Fanuc KAREL source: kb00151.KL

-- PROVISIONAL review KL for V940-1; original PC SHA256 d89378294aba81f9006a17e8a455f7a479b04fc5cfe738be1af26e2c5bc774eb
-- Incomplete behavior may be omitted. Consult companion uncertainty JSON. Do not deploy.
PROGRAM KB00151
%NOLOCKGROUP
BEGIN
  -- V9_ZERO_TABLE_METADATA_HINT layout=0002_ascii; no indexed target words; source/name/runtime held
  -- UNRESOLVED_PC offsets 5-14; opcodes 3F,75
  -- UNRESOLVED_PC offsets 19-26; opcodes 9D,23
  -- UNRESOLVED_PC offsets 31-38; opcodes 9D,23
  -- UNRESOLVED_PC offsets 43-73; opcodes 27,22,2A,22,22,22,31
  -- UNRESOLVED_PC offsets 78-82; opcodes 7F
END KB00151
